FUNCTION_BLOCK TOnTimer
VAR
    TON1 : TON;
END_VAR

METHOD Delay : BOOL
VAR_INPUT
    In : BOOL;
END_VAR
TON1(IN := In);
Delay := TON1.Q;
END_METHOD

METHOD FB_init : BOOL
VAR_INPUT
	bInitRetains : BOOL; // if TRUE, the retain variables are initialized (warm start / cold start)
	bInCopyCode : BOOL;  // if TRUE, the instance afterwards gets moved into the copy code (online change)
    PresetTime : LREAL; // seconds
END_VAR
TON1.PT := LREAL_TO_TIME(PresetTime * 1000);
END_METHOD

PROPERTY OutputState : BOOL
GET
OutputState := TON1.Q;
END_GET
END_PROPERTY

PROPERTY PresetTime : LREAL
GET
PresetTime := TIME_TO_LREAL(TON1.PT)/1000.0; // in seconds
END_GET
SET
TON1.PT := LREAL_TO_TIME(PresetTime * 1000);
END_SET
END_PROPERTY

METHOD Reset
TON1(IN := FALSE);
END_METHOD

METHOD Run : BOOL
TON1(IN := TRUE);
Run := TON1.Q;
END_METHOD

END_FUNCTION_BLOCK

(* stored: Version 1.1.0.1, ProductVersion 3.1.4024.3
   POU TOnTimer: Id {bd973412-bb37-46dd-8bca-85a58d3ce04e}, SpecialFunc None
   Method Delay: Id {d77dac6c-e6be-40f6-ba1e-301b376167b0}
   Method FB_init: Id {88d1c24e-7b16-4670-b38a-ca09f83895e8}
   Property OutputState: Id {7863916d-9ff4-0beb-2d0c-3a28d19b5791}
   Get Get: Id {6dc9f3b3-2d9f-0075-24b8-af5e17487166}
   Property PresetTime: Id {1f9fb480-1b12-4178-8125-c63f19e3f6c8}
   Get Get: Id {d9314860-65a5-469e-b7f4-05b64489e7a3}
   Set Set: Id {7421dbd3-c725-4152-b0f8-5a66f66ac11b}
   Method Reset: Id {10c74e56-67a0-476d-8779-307e14d54d6f}
   Method Run: Id {ae81aa91-5bbd-4d62-9bbb-8c0a060929be} *)
